(******************************************************************************
Baustein: FB_Testsuite
Spezifikation: doc/Spezifikation.pdf, Kap. x.y.z
-------------------------------------------------------------------------------
erstellt:
von:
Geändert:
von:
-------------------------------------------------------------------------------
Beschreibung
Dieser Baustein enthält alle zugeordneten Testfälle. Ein Testfall
ist ein abgeleiteter Baustein (FB) von FB_TestBase.

-------------------------------------------------------------------------------
Input
-

Output
-
******************************************************************************)
FUNCTION_BLOCK FB_Testsuite
    IMPLEMENTS ITestsuite_t
VAR_INPUT
END_VAR
VAR_OUTPUT
	o_eState  		: EState_t;
	o_eResult 		: EResult_t;
END_VAR
VAR
	strId			: ObjectId_t;
	strPath			: ObjectId_t;
	bRegistered     : BOOL;
	a_iTest  		: ARRAY [0..255] OF ITestBase_t;
	iTest     		: ITestBase_t;
	u16TestCases  	: UINT;
	u16Index 		: UINT;
	sStatistic 		: SStatistic_t;
END_VAR

(******************************************************************************
Baustein: FB_Testsuite.addTestcase
Spezifikation: doc/Spezifikation.pdf, Kap. x.y.z
-------------------------------------------------------------------------------
erstellt:
von:
Geändert:
von:
-------------------------------------------------------------------------------
Beschreibung
Diese Methode

-------------------------------------------------------------------------------
Input
i_pTestCase

Output
-
******************************************************************************)
{attribute 'hide'} 
METHOD PUBLIC addTestcase : BOOL
VAR_INPUT
	i_iTestCase : ITestBase_t;
END_VAR

	addTestcase := FALSE;

	IF 	i_iTestCase  <> 0   AND 
		u16TestCases <  255 THEN
		
		a_iTest[u16TestCases] := i_iTestCase;
		
		u16TestCases := u16TestCases +1;
		
		sStatistic.u32TestCases := sStatistic.u32TestCases + 1;
		
		addTestcase := true;
	END_IF
END_METHOD

METHOD execute : BOOL
VAR_INPUT
	i_bStart	: BOOL;
END_VAR
VAR
    sTestResult : STestcase_t;
END_VAR

	CASE o_eState OF
		
	EState_t.eStateInit:
	
		o_eState 	:= EState_t.eStateError;
		IF bRegistered = TRUE THEN
			o_eState 	:= EState_t.eStateIdle;
		END_IF;
		
	EState_t.eStateIdle:

		u16Index := 0;

		IF i_bStart = TRUE THEN
			logInfo(CONCAT('Run Testsuite ', strId));
			iTest 	 := getFirstTestCase();
			IF iTest <> 0 THEN
				logInfo(CONCAT('Execute Testcase ', iTest.getId()));
			END_IF;
			sStatistic.u32Executed  := 0;
			sStatistic.u32Passed 	:= 0;
			sStatistic.u32Failed 	:= 0;
			sStatistic.u32Asserts 	:= 0;
			o_eState  := EState_t.eStatePrepare;
			o_eResult := EResult_t.eStatePassed;
		END_IF;

	EState_t.eStatePrepare:

		IF iTest <> 0 THEN
			sTestResult := iTest.Result;
			IF sTestResult.eState <> EResult_t.eStateSkipped THEN
				 IF iTest._prepare() = ERetCode_t.eRetDone THEN
					  o_eState := EState_t.eStateExecute;
				 END_IF;
			ELSE
				 iTest 	:= getNextTestCase();
			END_IF;
		ELSE
			o_eState := EState_t.eStateREady;			
		END_IF;

	EState_t.eStateExecute:

		sTestResult := iTest.Result;

		IF iTest._execute()    = ERetCode_t.eRetDone		 	  OR 
			sTestResult.eState  = EResult_t.eStateFailedFatal THEN
			
			sStatistic.u32Executed := sStatistic.u32Executed + 1;	
			  (* update Result *)
			sTestResult := iTest.Result;
		
			sStatistic.u32Passed 	:= sStatistic.u32Passed + sTestResult.u32Passed;
			sStatistic.u32Failed 	:= sStatistic.u32Failed + sTestResult.u32Failed;
			sStatistic.u32Asserts   := sStatistic.u32Passed + sStatistic.u32Failed;
			
			// Status des aktuellen Tests auswerten
			CASE sTestResult.eState OF
			EResult_t.eStatePassed     : logInfo('	Test Passed');
			EResult_t.eStateFailed     : logInfo('	Test Failed');
			EResult_t.eStateFailedFatal: logInfo('	Test Failed Fatal');	
			END_CASE
			
			// Status der Testsuite ermitteln
			CASE o_eResult OF 

			EResult_t.eStatePassed:
				// Status des letzen Tests übernehmen
				o_eResult := sTestResult.eState;
				

			EResult_t.eStateFailed:
				// Status nur übernehmen wenn ein Fatal-Status
				// ermittelt wird und der Test sofort abgebrochen
				// werden soll.
				IF sTestResult.eState = EResult_t.eStateFailedFatal THEN
					o_eResult := sTestResult.eState;
					o_eState  := EState_t.eStateCleanUp;
				END_IF;		

			END_CASE;

			o_eState := EState_t.eStateCleanUp;

			IF o_eResult = EResult_t.eStateFailedFatal THEN
				o_eState := EState_t.eStateReady;					
			END_IF;

		END_IF;

	ESTate_t.eStateCleanUp:

		IF iTest <> 0 THEN
			IF iTest._cleanup() = ERetCode_t.eRetDone THEN
				iTest 	:= getNextTestCase();
				o_eState := EState_t.eStatePrepare;
			END_IF;
		ELSE
			o_eState := EState_t.eStateReady;
		END_IF;
		
	ESTate_t.eStateReady:
	
		IF i_bStart = FALSE THEN
			o_eState := EState_t.eStateIdle;
		END_IF
		
	ESTate_t.eStateError:	
		
		// wenn wir hier rauskommen ist was dummes passiert
		
	ELSE
		
		o_eState := EState_t.eStateError;
		
	END_CASE;
	
	
	
	
	
	
//
END_METHOD

(******************************************************************************
Baustein: FB_Testsuite.FB_init
Spezifikation: doc/Spezifikation.pdf, Kap. x.y.z
-------------------------------------------------------------------------------
erstellt:
von:
Geändert:
von:
-------------------------------------------------------------------------------
Beschreibung
Diese Methode

-------------------------------------------------------------------------------
Input
i_pTestCase

Output
-
******************************************************************************)
{attribute 'hide'} 
METHOD FB_init : BOOL
VAR_INPUT
	bInitRetains 	: BOOL; // if TRUE, the retain variables are initialized (warm start / cold start)
	bInCopyCode 	: BOOL;  // if TRUE, the instance afterwards gets moved into the copy code (online change)
	i_strId	  		: ObjectId_t;
	i_strPath		: ObjectId_t;
END_VAR

	strId 	:= i_StrId;
	strPath := i_strPath;
	register();
END_METHOD

(******************************************************************************
Baustein: FB_Testsuite.getFirstTestCase
Spezifikation: doc/Spezifikation.pdf, Kap. x.y.z
-------------------------------------------------------------------------------
erstellt:
von:
Geändert:
von:
-------------------------------------------------------------------------------
Beschreibung
Diese Methode

-------------------------------------------------------------------------------
Input
-

Output
-
******************************************************************************)
{attribute 'hide'} 
METHOD PUBLIC getFirstTestCase : ITestBase_t
VAR_INPUT
END_VAR

	u16Index := 0;
	getFirstTestCase := a_iTest[0];
END_METHOD

(******************************************************************************
Baustein: FB_Testsuite.getId
Spezifikation: doc/Spezifikation.pdf, Kap. x.y.z
-------------------------------------------------------------------------------
erstellt:
von:
Geändert:
von:
-------------------------------------------------------------------------------
Beschreibung
Diese Methode

-------------------------------------------------------------------------------
Input
-

Output
-
******************************************************************************)
{attribute 'hide'} 
METHOD PUBLIC getId : STRING
VAR_INPUT
END_VAR

	getId := strId;
END_METHOD

(******************************************************************************
Baustein: FB_Testsuite.getNextTestCase
Spezifikation: doc/Spezifikation.pdf, Kap. x.y.z
-------------------------------------------------------------------------------
erstellt:
von:
Geändert:
von:
-------------------------------------------------------------------------------
Beschreibung
Diese Methode

-------------------------------------------------------------------------------
Input
-

Output
-
******************************************************************************)
{attribute 'hide'} 
METHOD PUBLIC getNextTestCase : ITestBase_t
VAR_INPUT
END_VAR

	getNextTestCase := 0;
	u16Index 		 := u16Index + 1;

	IF u16Index < u16TestCases THEN
		getNextTestCase := a_iTest[u16Index];
	END_IF;
END_METHOD

{attribute 'hide'} 
METHOD PUBLIC getPath : ObjectId_t
VAR_INPUT
END_VAR

	getPath := strPath;
END_METHOD

METHOD getResult : EResult_t
VAR_INPUT
END_VAR

	getResult := o_eResult;
END_METHOD

METHOD getState : EState_t
getState := o_eState;
END_METHOD

(******************************************************************************
Baustein: FB_Testsuite.logInfo
Spezifikation: doc/Spezifikation.pdf, Kap. x.y.z
-------------------------------------------------------------------------------
erstellt:
von:
Geändert:
von:
-------------------------------------------------------------------------------
Beschreibung
Diese Methode

-------------------------------------------------------------------------------
Input
i_strMessage

Output
-
******************************************************************************)
{attribute 'hide'} 
METHOD PROTECTED logInfo : BOOL
VAR_INPUT
	i_strMessage : StrMessage_t;
END_VAR

	ADSLOGSTR(msgCtrlMask 	:= ADSLOG_MSGTYPE_HINT , 
			  msgFmtStr 	:= i_strMessage, 
			  strArg 		:= '');
END_METHOD

(******************************************************************************
Baustein: FB_Testsuite.register
Spezifikation: doc/Spezifikation.pdf, Kap. x.y.z
-------------------------------------------------------------------------------
erstellt:
von:
Geändert:
von:
-------------------------------------------------------------------------------
Beschreibung
Diese Methode

-------------------------------------------------------------------------------
Input
-

Output
-
******************************************************************************)
{attribute 'hide'} 
METHOD PROTECTED register : BOOL
VAR_INPUT
END_VAR

	bRegistered := PRG_TestLib.addTestSuite(this^);
END_METHOD

{warning 'Eigenschaftenimplementierung hinzufügen'}
PROPERTY Result : SStatistic_t
GET
Result := sStatistic;
END_GET
END_PROPERTY

END_FUNCTION_BLOCK

(* stored: Version 1.1.0.1, ProductVersion 3.1.4024.12
   POU FB_Testsuite: Id {ae8bbd51-73a9-4be0-b082-2ec8a068e7f6}, SpecialFunc None
   Method addTestcase: Id {80822225-6192-4f00-bbb8-24a92c6881f7}
   Method execute: Id {44c9852e-be60-482d-af64-b35cb0a07d5a}
   Method FB_init: Id {cdfd5773-6fa2-4b78-87a3-142799abac6a}
   Method getFirstTestCase: Id {565a7440-2552-4228-bd2b-b6378bb5c8b9}
   Method getId: Id {f75a7191-de66-4010-8dda-4a26aa6a90f4}
   Method getNextTestCase: Id {caddd296-a017-4642-872a-27f49eaad75c}
   Method getPath: Id {0c655e80-1810-4039-ac18-fb19e58b187c}
   Method getResult: Id {da61837f-a28c-4b0f-93ef-935f7efb76a4}
   Method getState: Id {043e226a-4a17-4c00-b80f-6dbe5fb3b88f}
   Method logInfo: Id {4162b475-e111-4ea4-af72-09599d7cdb23}
   Method register: Id {3a42094d-f3f7-40aa-9e2e-e1eb00f9e432}
   Property Result: Id {a498e662-1794-43fc-873e-a36fb9fd250b}
   Get Get: Id {55f23317-ab5c-4ecf-9850-69ee41479e24} *)
